FUNCTION_BLOCK Payload_Carrier 
VAR_INPUT
END_VAR
VAR_OUTPUT
END_VAR
VAR
	aPayloads : ARRAY[1..PAYLOAD_TYPE_SIZE-1] OF I_Payload;
	//iPayload : I_Payload;
	ePayloadType : E_Payload_Type;
END_VAR

METHOD GetPayload : BOOL
VAR_IN_OUT
	pByte : POINTER TO BYTE;
END_VAR

VAR_INPUT
	ePayloadType : E_Payload_Type;
END_VAR
(*
IF 	THIS^.ePayloadType = ePayloadType
	THEN
		GetPayload :=  __QUERYPOINTER(iPayload, pByte);
END_IF
*)


IF 	aPayloads[ePayloadType] <> 0
	THEN
		GetPayload :=  __QUERYPOINTER(aPayloads[ePayloadType], pByte);
END_IF
END_METHOD

METHOD SetPayload : BOOL
VAR_INPUT
	iPayload : I_Payload; 
	ePayloadType : E_Payload_Type;
END_VAR
(*
IF ePayloadType <> NO_PAYLOAD
	THEN
	
	THIS^.iPayload := iPayload;
	THIS^.ePayloadType := ePayloadType;
	
	SetPayload := TRUE;
	
END_IF
*)

IF ePayloadType <> NO_PAYLOAD
	THEN
	
	THIS^.aPayloads[ePayloadType] := iPayload;
	
	SetPayload := TRUE;
	
END_IF
END_METHOD

END_FUNCTION_BLOCK

(* stored: Version 1.1.0.1, ProductVersion 3.1.4024.2
   POU Payload_Carrier: Id {1fa36593-3ecc-43fd-a15b-6576771ee199}, SpecialFunc None
   Method GetPayload: Id {529fe2e9-48db-47b1-b9db-042c523f458f}
   Method SetPayload: Id {1ada05a6-5913-4254-88a8-7e46ea56218a} *)
